INTERFACE ITF_PB_Element EXTENDS __SYSTEM.IQueryInterface

PROPERTY PUBLIC P_DisableAxis12 : BOOL
SET
END_SET
END_PROPERTY

PROPERTY PUBLIC P_EmuSpeed : INT
SET
END_SET
END_PROPERTY

PROPERTY PUBLIC P_RegisterFuncton : PVOID
GET
END_GET
SET
END_SET
END_PROPERTY

END_INTERFACE

(* stored: Version 1.1.0.1, ProductVersion 3.1.4024.9
   Itf ITF_PB_Element: Id {fa2b6137-22b8-487e-9b45-0b34c434ee11}
   Property P_DisableAxis12: Id {add6aa3c-f5b8-4e7a-bfb5-048c5a43263e}
   Set Set: Id {83774731-1cd7-4235-bb19-91780f867a92}
   Property P_EmuSpeed: Id {64397e0a-0a25-4855-9402-fd3fac618dea}
   Set Set: Id {5b7704bc-56ef-44e8-845a-ba40e2b91e71}
   Property P_RegisterFuncton: Id {c40bc93f-1631-4b16-ba95-d22721ca5b66}
   Get Get: Id {cb093a35-fbda-46b8-8083-7144ae06e9af}
   Set Set: Id {dc867f87-c0d3-4c6e-88e8-991426820f33} *)
